Staubli VAL3: onRun.pgx

public program onRun(string& x_sItem[])
  local string l_sEmpty
  local num l_nResult
  local num l_nIndex
  local mdesc l_mDesc
  local bool l_bUnreached
  local num l_nMoveId
  local string l_sComment
  local Trajectory l_tTraj
  local joint l_jJoint
begin
  if find(x_sItem,"@HOME")!=-1
    //load the home home
    l_nResult=home:libLoad(saveData:sPathTraj+"HOME")
    delay(0)
    l_nIndex=size(home:tTraj["home"].tData)-1
    l_mDesc=home:tTraj["home"].tData[l_nIndex].tSuper.nom_speed
    l_jJoint=home:tTraj["home"].tData[l_nIndex].jJoint
    // execute the movement
    call moveTo(flange,l_mDesc,0,l_bUnreached,l_jJoint,l_nMoveId)
    // show the comments
    l_tTraj.tSuper=home:tTraj["home"].tData[l_nIndex].tSuper
    l_tTraj.sID="JPOINT @HOME"
    call cycleStatus:addTraj(l_tTraj)
    wait(getMoveId()>=l_nMoveId-0.1 or isEmpty())
  else
    // execute check if need to reload
    call loadCycle(x_sItem,l_nResult)
    if l_nResult==0
      // execute
      call makeTraj(x_sItem)
    else
      popUpMsg("JOINT NOT DEFINE !!!")
      cycleStatus:bToStop=false
    endIf
  endIf
end
